# EPICS substitutions: mks647c.substitutions
file mks647c.template
{
pattern {S, TA, DN, DT1, DT2}
        {BL11A, SE, mks647c, MF, PR}
}
